// TIA Portal V20 export
ORGANIZATION_BLOCK "Startup"   // OB1000, LAD, Startup
TITLE = "Complete Restart"
AUTHOR : ERsystem_FA2_DH. Kim
// stored: AutoNumber false, IsIECCheckEnabled true, Namespace Unit1, SetENOAutomatically false
   VAR_INPUT
      LostRetentive : Bool;   // True if retentive data are lost
      LostRTC : Bool;   // True if date and time are lost
   END_VAR
   VAR_TEMP
      tempIndex : Int;   // Index of Unit in the array
   END_VAR
BEGIN

REGION Network 1: Unit Index Number
   // Assign the number of the unit to a temp for correct array index access.
   // Number is defined in PLC tags of Software Unit Global.
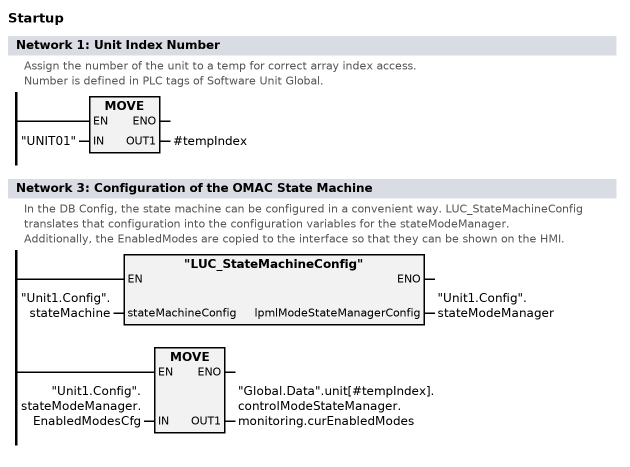
   RUNG wire#powerrail
      Move(in := "UNIT01", out1 => #tempIndex)
   END_RUNG
   // the same network as SCL:
   #tempIndex := "UNIT01";
END_REGION

REGION Network 2 (SCL): Build the Absolut Reference Designator
   // Set the Absoult Reference Designator in the DB Config. It is combined out of the parent reference designator and the own reference designator (=relative)
   IF LEN(IN := "Unit1.Config".unit.referenceDesignator.parent) <> 0 THEN
     "Unit1.Config".unit.referenceDesignator.combined := CONCAT_WSTRING(IN1 := "Unit1.Config".unit.referenceDesignator.parent, IN2 := WSTRING#'.', IN3 := "Unit1.Config".unit.referenceDesignator.relative);
   ELSE
     "Unit1.Config".unit.referenceDesignator.combined := "Unit1.Config".unit.referenceDesignator.relative;
   END_IF;
END_REGION

REGION Network 3: Configuration of the OMAC State Machine
   // In the DB Config, the state machine can be configured in a convenient way. LUC_StateMachineConfig translates that configuration into the configuration variables for the stateModeManager.
   // Additionally, the EnabledModes are copied to the interface so that they can be shown on the HMI.
   RUNG wire#powerrail
      "LUC_StateMachineConfig"(stateMachineConfig := "Unit1.Config".stateMachine, lpmlModeStateManagerConfig => "Unit1.Config".stateModeManager)
   END_RUNG
   RUNG wire#powerrail
      Move(in := "Unit1.Config".stateModeManager.EnabledModesCfg, out1 => "Global.Data".unit[#tempIndex].controlModeStateManager.monitoring.curEnabledModes)
   END_RUNG
   // the same network as SCL:
   "LUC_StateMachineConfig"(stateMachineConfig := "Unit1.Config".stateMachine,
                           lpmlModeStateManagerConfig => "Unit1.Config".stateModeManager);
   "Global.Data".unit[#tempIndex].controlModeStateManager.monitoring.curEnabledModes := "Unit1.Config".stateModeManager.EnabledModesCfg;
END_REGION
END_ORGANIZATION_BLOCK
